// TIA Portal project "项目2" (V16)

(* hardware
DEVICE "S7-1200 station_2"  S7-1200 Station
   slot 0: "Rack_0"  S7-1200 Rack  Rack  V1.0
   slot 1: "PLC_2"  CPU 1212C DC/DC/DC  6ES7 212-1AE40-0XB0  V4.4
DEVICE "S7-1200 station_1"  S7-1200 Station
   slot 0: "Rack_0"  S7-1200 Rack  Rack  V1.0
   slot 1: "PLC_1"  CPU 1214C DC/DC/DC  6ES7 214-1AG40-0XB0  V4.4
DEVICE "HMI_1"  KTP700 Basic PN Portrait
   slot 0: "HMI_1"  KTP700 Basic PN Portrait  6AV2 123-2GB03-0AX0  16.0.0.0
   slot 1: "HMI_RT_1"  KTP700 Basic PN Portrait  6AV2 123-2GB03-0AX0  16.0.0.0
   slot 5: "HMI_1.IE_CP_1"  PROFINET Interface  16.0.0.0
      slot 1: "PROFINET Interface_1"  PROFINET Interface
         slot 1: "Port_1"  Port
*)

// ===== PLC "PLC_1"  CPU 1214C DC/DC/DC =====

VAR_GLOBAL   // PLC tag table "默认变量表"
   "Clock_Byte" AT %MB0 : Byte;
   "Clock_10Hz" AT %M0.0 : Bool;
   "Clock_5Hz" AT %M0.1 : Bool;
   "Clock_2.5Hz" AT %M0.2 : Bool;
   "Clock_2Hz" AT %M0.3 : Bool;
   "Clock_1.25Hz" AT %M0.4 : Bool;
   "Clock_1Hz" AT %M0.5 : Bool;
   "Clock_0.625Hz" AT %M0.6 : Bool;
   "Clock_0.5Hz" AT %M0.7 : Bool;
   "System_Byte" AT %MB1 : Byte;
   "FirstScan" AT %M1.0 : Bool;
   "DiagStatusUpdate" AT %M1.1 : Bool;
   "AlwaysTRUE" AT %M1.2 : Bool;
   "AlwaysFALSE" AT %M1.3 : Bool;
END_VAR

DATA_BLOCK "发送DB"   // DB1
{ S7_Optimized_Access := 'FALSE' }
VERSION : 0.1
   VAR
      发送 : Struct
         发信号 : Array[0..20] of Byte;
      END_STRUCT;
   END_VAR
BEGIN
END_DATA_BLOCK

DATA_BLOCK "数据块_1"   // DB4
{ S7_Optimized_Access := 'TRUE' }
VERSION : 0.1
   VAR
      qid : Bool;
   END_VAR
BEGIN
END_DATA_BLOCK

// folder: System blocks/Program resources

DATA_BLOCK "PLC_1_Send_DB"   // DB3
{ S7_Optimized_Access := 'TRUE' }
AUTHOR : SIMATIC
FAMILY : MC7Plus
NAME : TC_IP_v4
VERSION : 1.0
// stored: InstanceOfName TCON_IP_v4
"TCON_IP_v4"
BEGIN
   ID := 1;
   InterfaceId := 64;
   RemotePort := 2000;
   ActiveEstablished := true;
   RemoteAddress.ADDR[1] := 192;
   RemoteAddress.ADDR[2] := 168;
   RemoteAddress.ADDR[4] := 2;
END_DATA_BLOCK

// folder: (top level)

ORGANIZATION_BLOCK "Main"   // OB1, LAD, ProgramCycle
TITLE = "Main Program Sweep (Cycle)"
{ S7_Optimized_Access := 'TRUE' }
VERSION : 0.1
   VAR_INPUT
      Initial_Call : Bool;   // Initial call of this OB
      Remanence : Bool;   // =True, if remanent data are available
   END_VAR
BEGIN

REGION Network 1: 用来发送
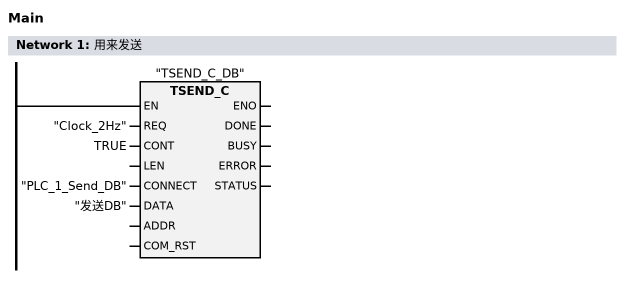
   "TSEND_C_DB"(REQ := "Clock_2Hz", CONT := TRUE, CONNECT := "PLC_1_Send_DB", DATA := "发送DB");   // TSEND_C
END_REGION
END_ORGANIZATION_BLOCK

// ===== PLC "PLC_2"  CPU 1212C DC/DC/DC =====

VAR_GLOBAL   // PLC tag table "默认变量表"
   "System_Byte" AT %MB1 : Byte;
   "FirstScan" AT %M1.0 : Bool;
   "DiagStatusUpdate" AT %M1.1 : Bool;
   "AlwaysTRUE" AT %M1.2 : Bool;
   "AlwaysFALSE" AT %M1.3 : Bool;
   "Clock_Byte" AT %MB0 : Byte;
   "Clock_10Hz" AT %M0.0 : Bool;
   "Clock_5Hz" AT %M0.1 : Bool;
   "Clock_2.5Hz" AT %M0.2 : Bool;
   "Clock_2Hz" AT %M0.3 : Bool;
   "Clock_1.25Hz" AT %M0.4 : Bool;
   "Clock_1Hz" AT %M0.5 : Bool;
   "Clock_0.625Hz" AT %M0.6 : Bool;
   "Clock_0.5Hz" AT %M0.7 : Bool;
END_VAR

DATA_BLOCK "接受DB块"   // DB1
{ S7_Optimized_Access := 'FALSE' }
VERSION : 0.1
   VAR
      接收 : Struct
         接信号 : Array[0..20] of Byte;
      END_STRUCT;
   END_VAR
BEGIN
END_DATA_BLOCK

// folder: System blocks/Program resources

DATA_BLOCK "PLC_2_Receive_DB"   // DB3
{ S7_Optimized_Access := 'TRUE' }
AUTHOR : SIMATIC
FAMILY : MC7Plus
NAME : TC_IP_v4
VERSION : 1.0
// stored: InstanceOfName TCON_IP_v4
"TCON_IP_v4"
BEGIN
   ID := 1;
   InterfaceId := 64;
   LocalPort := 2000;
   RemoteAddress.ADDR[1] := 192;
   RemoteAddress.ADDR[2] := 168;
   RemoteAddress.ADDR[4] := 1;
END_DATA_BLOCK

// folder: (top level)

ORGANIZATION_BLOCK "Main"   // OB1, LAD, ProgramCycle
TITLE = "Main Program Sweep (Cycle)"
{ S7_Optimized_Access := 'TRUE' }
VERSION : 0.1
   VAR_INPUT
      Initial_Call : Bool;   // Initial call of this OB
      Remanence : Bool;   // =True, if remanent data are available
   END_VAR
BEGIN

REGION Network 1
   // 接受1214的数据，存到DB1212中
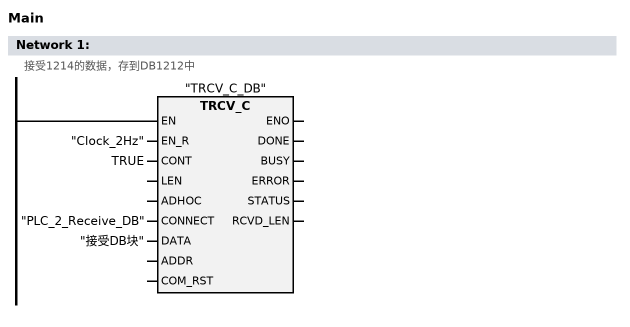
   "TRCV_C_DB"(EN_R := "Clock_2Hz", CONT := TRUE, CONNECT := "PLC_2_Receive_DB", DATA := "接受DB块");   // TRCV_C
END_REGION
END_ORGANIZATION_BLOCK

(* ===== HMI "HMI_RT_1" =====
system functions are stored by id; their names below are inferred from use
connection "HMI_连接_1": ETHERNET, SMART_S7_1200_OMS

HMI tags "默认变量表"
   "Tag_ScreenNumber" : UInt, internal
   "发送DB_发送_发信号{0}" : Byte = PLC 发送DB.发送.发信号[0] AT %DB1.DBB0, 1 s

discrete alarms
   2: '正在计时', class Errors, trigger "Tag_ScreenNumber" bit 0

Template "模板_1" 480x800
   Button "起始画面" at 428,61 size 50x71; TextOff '起始画面'; PictureOff "NavigateHome_KTP700_Basic_PN_Portrait_TR"; PictureOn "NavigateHome_KTP700_Basic_PN_Portrait_TR"
      on Release: ActivateScreen("根画面", 0)
   Button "Template_Button" at 428,172 size 50x71; TextOff 'Text'
   Button "Template_Button_1" at 428,283 size 50x71; TextOff 'Text'
   Button "Template_Button_2" at 428,394 size 50x71; TextOff 'Text'
   Button "Template_Button_3" at 428,505 size 50x71; TextOff 'Text'
   Button "Template_Button_4" at 428,616 size 50x71; TextOff 'Text'
   Button "退出" at 428,727 size 50x71; TextOff '退出'; PictureOff "ExitRuntime_KTP700_Basic_PN_Portrait_TR"; PictureOn "ExitRuntime_KTP700_Basic_PN_Portrait_TR"
      on Release: StopRuntime(0)
   SymbolicIOField "Symbolic_IO_Field_Screen" at 109,11 size 264x38; TextOff '0'; TextOn '1'; TextList "TextList_ScreenNames"
      ProcessValue <- "Tag_ScreenNumber"
      on Change: ActivateScreenByNumber("Tag_ScreenNumber", 0)
   DateTimeField "HmiScreenItemData" at 375,30 size 105x30
   DateTimeField "HmiScreenItemData_1" at 375,0 size 105x30
   GraphicView "Logo" at 0,0 size 107x60; Picture "HMI_1 的 Logo"

screen "根画面" 480x800, template "模板_1"
   on GenerateScreen: SetTag("Tag_ScreenNumber", 1)
   Button "按钮_1" at 127,146 size 96x32; TextOff 'Text'
      on Click: ActivateScreen("画面_1", 0)
*)